{attribute 'qualified_only'}
{attribute 'strict'}
{attribute 'to_string'}
TYPE S7_COMMUNICATOR_STATE :
(
	IDLE_OR_DONE,
	DATA_PROCESSING,
	WAIT_FOR_NEXT_CYCLE
);
END_TYPE

(* stored: Version 1.1.0.1
   DUT S7_COMMUNICATOR_STATE: Id {485eded7-31f1-0c06-3d02-ac21e0382df7} *)
